Fanuc KAREL source: kt00189.KL

PROGRAM KT00189
%NOLOCKGROUP
VAR
H1 : ARRAY[2] OF SHORT
Y2 : ARRAY[2] OF BYTE
OUT:INTEGER
BEGIN
H1[1]=2
Y2[1]=3
OUT=(H1[1] MOD Y2[1])
END KT00189
